(* PLC project  *)

CONFIGURATION Empty_Module_12
END_CONFIGURATION
